FUNCTION_BLOCK Spray
VAR_INPUT
	bExecute:BOOL;
	Order:ARRAY[0..7] OF INT;//世界坐标系下的夹具次序
	Angle:REAL;
END_VAR
VAR_OUTPUT
	bDone: BOOL;
END_VAR
VAR
	pick:INT;
	SpraySwitch:ARRAY[0..7] OF BOOL:=[0,0,0,0,0,0,0,0];//Order by Eletronic
	SwitchOpen:ARRAY[0..7] OF INT:=[0,0,0,0,0,0,0,0];//Order by Eletronic
	Angle2Switch:ARRAY[0..7] OF INT:=[3,2,1,8,7,6,5,4];
	SensorSignal:BOOL:=TRUE;
	i: INT;
END_VAR

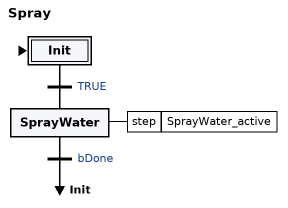
INITIAL_STEP Init:
END_STEP
TRANSITION FROM Init TO SprayWater
    := TRUE;
END_TRANSITION
STEP SprayWater:
    SprayWater_active(N);  // step action
END_STEP
TRANSITION FROM SprayWater TO Init
    := bDone;
END_TRANSITION

ACTION SprayWater_active:
pick:= REAL_TO_INT(Angle/(-45));
IF pick = 8 THEN
	pick:=0;
END_IF
IF SensorSignal THEN
	//By Order
	//SpraySwitch[Order[2]-1]:=TRUE;
	//SwitchOpen[Order[2]-1]:=SwitchOpen[Order[2]-1]+1;
	//By Angle
	SpraySwitch[Angle2Switch[pick]-1]:=TRUE;
	SwitchOpen[Angle2Switch[pick]-1]:=SwitchOpen[Angle2Switch[pick]-1]+1;
END_IF
SensorSignal:=FALSE;
//SpraySwitch[Order[3]-1]:=FALSE;

IF pick=0 THEN
	SpraySwitch[Angle2Switch[7]-1]:=FALSE;
	SwitchOpen[Angle2Switch[7]-1]:=0;
ELSE
	SpraySwitch[Angle2Switch[pick-1]-1]:=FALSE;
	SwitchOpen[Angle2Switch[pick-1]-1]:=0;
END_IF

FOR i := 0 TO 7 DO
	IF SwitchOpen[i]>=20 THEN
		SpraySwitch[i]:=FALSE;
		SwitchOpen[i]:=0;
	END_IF
END_FOR
END_ACTION

END_FUNCTION_BLOCK

(* stored: Version 1.1.0.1, ProductVersion 3.1.4024.12
   POU Spray: Id {c22f7627-87e4-479a-a730-a9acd11ec63e}, SpecialFunc None
   Action SprayWater_active: Id {1791eb3e-3b90-4a2d-a9e0-9a6bee8902fe} *)
